// TwinCAT 3 PLC project Untitled1
// ProgramVersion: 3.1.4024.0
// libraries:
//   Tc2_Standard, * (Beckhoff Automation GmbH)
//   Tc2_System, * (Beckhoff Automation GmbH)
//   Tc3_Module, * (Beckhoff Automation GmbH)
// project tree:
//   DUTs/ dt_demo.TcDUT
//   / PlcTask.TcTTO
//   POUs/ MAIN.TcPOU
// real-time tasks:
//   TASK PlcTask: cycle T#10ms, priority 20, ADS port 350

CONFIGURATION Untitled1
    RESOURCE PLC ON TwinCAT3
        TASK PlcTask(INTERVAL := T#10ms, PRIORITY := 20);
        PROGRAM MAIN WITH PlcTask : MAIN;
    END_RESOURCE
END_CONFIGURATION

// ---- DUTs/dt_demo.TcDUT
TYPE dt_demo :
STRUCT
	on	: BOOL;
	cnt	: INT;
END_STRUCT
END_TYPE

// ---- POUs/MAIN.TcPOU
PROGRAM MAIN
VAR
	a	: dt_demo;
	b	: dt_demo;
	arr	: ARRAY[0..arr_max] OF dt_demo;
	i	: INT;
END_VAR
VAR CONSTANT
	arr_max	: INT := 1;
END_VAR


IF a.on THEN
	a.cnt := a.cnt + 1;
END_IF

IF b.on THEN
	b.cnt := b.cnt + 1;
END_IF

FOR i := 0 TO arr_max DO
	IF arr[i].on THEN
		arr[i].cnt := arr[i].cnt + 1;
	END_IF
END_FOR

END_PROGRAM
